(* Logix 5000 project; controller cal1615 1756-L62 rev 16.20; software revision 16.05; part 48 of 78 *)
(* tags used below, declared in another part *)
   FAULT : BOOL;   // Fault AFI
   p01_param_min_start_tension : REAL;
   p01_recipe_active : recipe;   // Active Recipe
   p01r02_plc_scan_time_in_sec : REAL;   // System PLC Scan Time in Seconds
   p01r09_pb_global_reset : BOOL;   // System Modes PB: Global Fault Reset
   p01r09_request_line_jog : BOOL;   // System Modes Request Line Jog Forward
   p01r09_stretch_mode : BOOL;
   p01r12_master_ramped_speed : REAL;   // System Line Accel Decel Control Master Ramped Speed
   p01r13_line_running : BOOL;   // System Line Start Sequence Line Running
   p01r13_line_slow_ramp : BOOL;   // System Line Start Sequence Start Line to Slow Speed
   p01r13_permissive_drives : BOOL;   // System Line Start Sequence Permissive Drives
   p01r13_state : DINT;   // System Line Start Sequence Sequencer Step
   p02_real_from_hmi : hmi_real;   // MOP HMI Iface Real from HMI
   p20r15_loa_on : BOOL;   // Letoff Letoff A VFD On
   p20r16_lob_on : BOOL;   // Letoff Letoff B On
   p22_ai_speed : REAL;
   p22_ai_ts1_lc : REAL;   // Tension Stand 1 Analog Input Loadcell
   p22_ao_selected_speed : REAL;   // Tension Stand 1 VFD Selected Speed
   p22_ao_torque : REAL;
   p22_control_word : INT;
   p22_di_brake : BOOL;   // Tension Stand 1 Digital Input Brake Temperature OK
   p22_di_jog : BOOL;   // Tension Stand 1 Digital Input SS: Jog
   p22_di_jog_fwd : BOOL;   // Tension Stand 1 Digital Input PB: Jog Forward
   p22_di_jog_rev : BOOL;   // Tension Stand 1 Digital Input PB: Jog Reverse
   p22_di_run : BOOL;   // Tension Stand 1 Digital Input SS: Run
   p22_di_therm : BOOL;   // Tension Stand 1 Digital Input Motor Temperature OK
   p22_param_ts1_jog_speed : REAL;   // System Parameter Tension Stand 1 Jog Speed
   p22_status_word : INT;
   p22_ts1_acc_rate : REAL;
   p22_ts1_decel_rate : REAL;
   p22_ts1_vfd : ABB_PROTOCOL_VFD;
   p22r01 : routine;   // Tension Stand 1 Main
   p22r02_tension_dev_max : REAL;   // Winder A VFD
   p22r02_tension_dev_min : REAL;   // Tension Stand 1 VFD
   p22r09 : routine;   // Tension Stand 1 Modes
   p22r09_mode_jog : BOOL;   // Tension Stand 1 Modes Jog Mode
   p22r09_mode_run : BOOL;   // Tension Stand 1 Modes Run Mode
   p22r09_mode_thread : BOOL;   // Tension Stand 1 Modes Thread Mode
   p22r09_pb_jog_fwd : BOOL;   // Tension Stand 1 Modes PB: Jog Forward
   p22r09_pb_jog_rev : BOOL;   // Tension Stand 1 Modes PB: Jog Reverse
   p22r09_timer_fault : TIMER[4];   // Tension Stand 1 Modes Fault Delay
   p22r09_timer_warning : TIMER[4];   // Tension Stand 1 Modes Warning Delay
   p22r10 : routine;   // Tension Stand 1 Speed Tension
   p22r10_calc_speed_offset : REAL;
   p22r10_param_psn_gain : REAL;   // Tension Stand 1 Parameter Position Gain
   p22r10_pid_out : REAL;
   p22r10_pid_psn : PID;   // Tension Stand 1 Speed Tension PID Dancer Position
   p22r10_pid_psn_cv : REAL;   // Tension Stand 1 Speed Tension PID Dancer Position Control Variable
   p22r10_pid_psn_pv : REAL;   // Tension Stand 1 Speed Tension PID Dancer Position Process Variable
   p22r10_selected_torque : REAL;
   p22r10_speed_offset : REAL;   // Tension Stand 1 Speed tension Speed Offset from Base
   p22r10_stretch : REAL;
   p22r10_timer_fault : TIMER[4];   // Tension Stand 1 Speed Tension Fault Delay
   p22r10_timer_warning : TIMER[4];   // Tension Stand 1 Speed Tension Warning Delay
   p22r11 : routine;   // Tension Stand 1 VFD
   p22r11_acc_decel_ramp : SYS_ACC_DEC_RAMP;   // Tension Stand 1 VFD Accel/Decel Ramp
   p22r11_permissive_jog : BOOL;   // Tension Stand 1 VFD Permissive Run
   p22r11_request_jog_fwd : BOOL;   // Tension Stand 1 VFD Request Jog FWD
   p22r11_request_jog_rev : BOOL;   // Tension Stand 1 VFD Request Jog REV
   p22r11_request_line_jog : BOOL;   // Tension Stand 1 VFD Request Line Jog
   p22r11_request_line_run : BOOL;   // Tension Stant 1 VFD Request Line Run
   p22r11_request_start : BOOL;   // Tension Stand 1 VFD
   p22r11_request_tension : BOOL;
   p22r11_request_thread_fwd : BOOL;   // Tension Stand 1 VFD Request Thread FWD
   p22r11_request_thread_rev : BOOL;   // Tension Stand 1 VFD Request Thread REV
   p22r11_selected_speed : REAL;   // Tension Stand 1 VFD Selected Speed
   p22r11_timer_fault : TIMER[10];   // Tension Stand 1 VFD Fault Timer
   p22r11_timer_warning : TIMER[5];   // Tension Stand 1 VFD Warning Timer
   p22r11_zero_speed : BOOL;   // Tension Stand 1 VFD Zero Speed
   p23r15_pid_tension_control : BOOL;   // Impreg Metering Roll VFD PID Wet Web Active
   p25r09_mode_thread : BOOL;   // Tension Stand 2 Modes Thread Mode
   p25r09_pb_jog_fwd : BOOL;   // Tension Stand 2 Modes PB: Jog Forward
   p25r09_pb_jog_rev : BOOL;   // Tension Stand 2 Modes PB: Jog Reverse
(* P22_Tension_Stand_1, continued *)

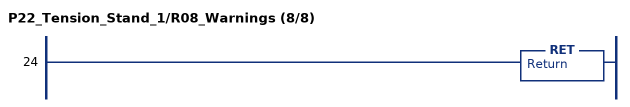
   [picture p936: P22_Tension_Stand_1/R08_Warnings rungs 24-24]
   24: RET();
END_ROUTINE

ROUTINE R09_Modes   (* ladder *)
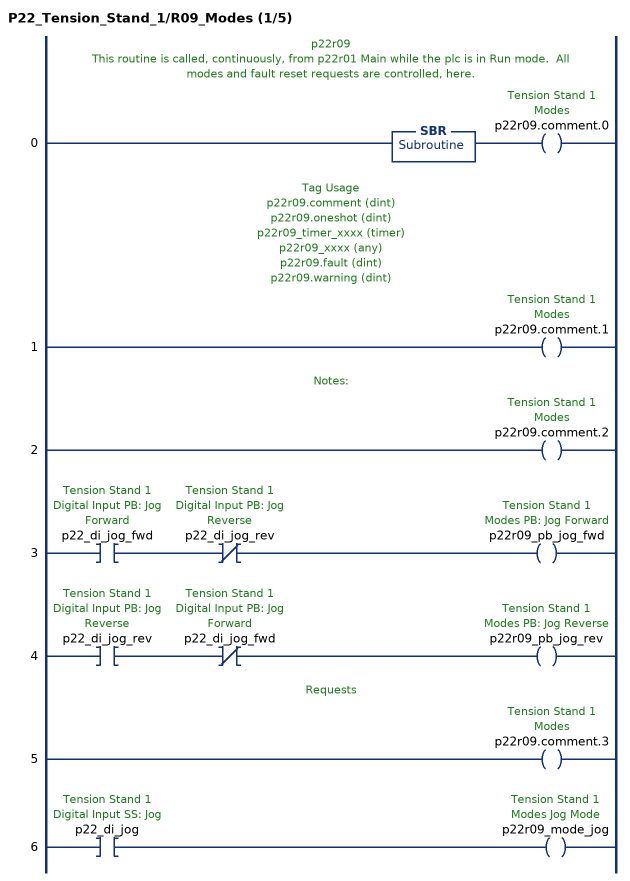
   // p22r09
   // This routine is called, continuously, from p22r01 Main while the plc is in Run mode.  All modes and fault reset requests are controlled, here.
   0: SBR()OTE(p22r09.comment.0);
   // Tag Usage
   // p22r09.comment (dint)
   // p22r09.oneshot (dint)
   // p22r09_timer_xxxx (timer)
   // p22r09_xxxx (any)
   // p22r09.fault (dint)
   // p22r09.warning (dint)
   1: OTE(p22r09.comment.1);
   // Notes:
   2: OTE(p22r09.comment.2);
   3: XIC(p22_di_jog_fwd)XIO(p22_di_jog_rev)OTE(p22r09_pb_jog_fwd);
   4: XIC(p22_di_jog_rev)XIO(p22_di_jog_fwd)OTE(p22r09_pb_jog_rev);
   // Requests
   5: OTE(p22r09.comment.3);
   6: XIC(p22_di_jog)OTE(p22r09_mode_jog);
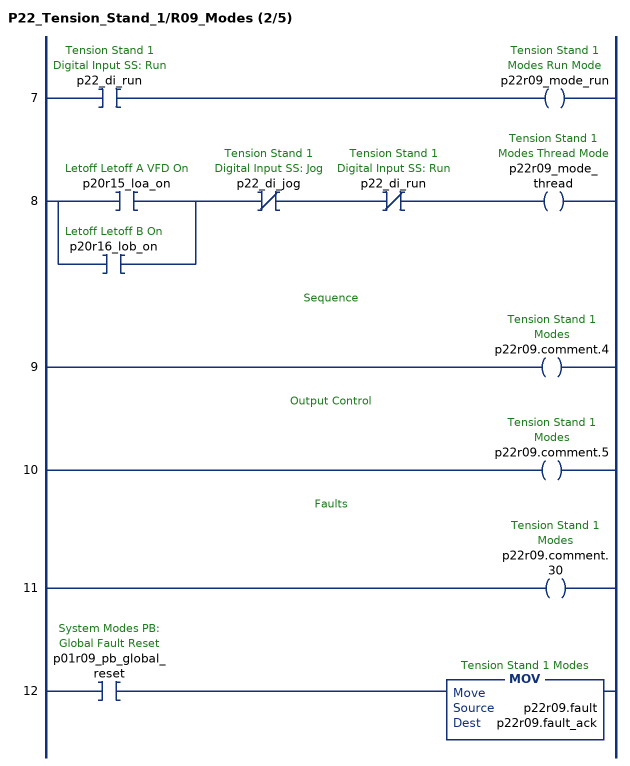
   7: XIC(p22_di_run)OTE(p22r09_mode_run);
   8: [XIC(p20r15_loa_on) ,XIC(p20r16_lob_on) ]XIO(p22_di_jog)XIO(p22_di_run)OTE(p22r09_mode_thread);
   // Sequence
   9: OTE(p22r09.comment.4);
   // Output Control
   10: OTE(p22r09.comment.5);
   // Faults
   11: OTE(p22r09.comment.30);
   12: XIC(p01r09_pb_global_reset)MOV(p22r09.fault,p22r09.fault_ack);
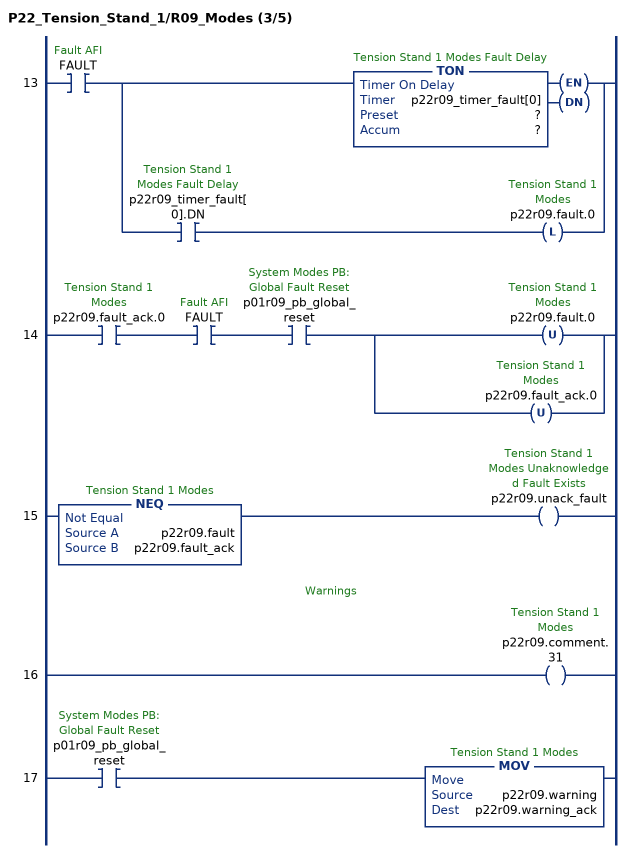
   13: XIC(FAULT)[TON(p22r09_timer_fault[0],?,?) ,XIC(p22r09_timer_fault[0].DN) OTL(p22r09.fault.0) ];
   14: XIC(p22r09.fault_ack.0)XIC(FAULT)XIC(p01r09_pb_global_reset)[OTU(p22r09.fault.0) ,OTU(p22r09.fault_ack.0) ];
   15: NEQ(p22r09.fault,p22r09.fault_ack)OTE(p22r09.unack_fault);
   // Warnings
   16: OTE(p22r09.comment.31);
   17: XIC(p01r09_pb_global_reset)MOV(p22r09.warning,p22r09.warning_ack);
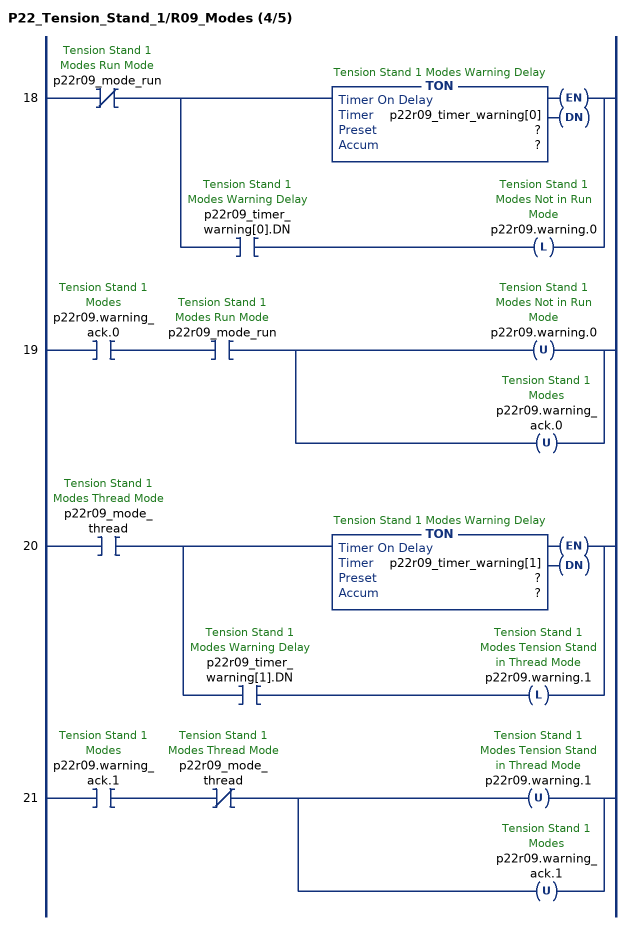
   18: XIO(p22r09_mode_run)[TON(p22r09_timer_warning[0],?,?) ,XIC(p22r09_timer_warning[0].DN) OTL(p22r09.warning.0) ];
   19: XIC(p22r09.warning_ack.0)XIC(p22r09_mode_run)[OTU(p22r09.warning.0) ,OTU(p22r09.warning_ack.0) ];
   20: XIC(p22r09_mode_thread)[TON(p22r09_timer_warning[1],?,?) ,XIC(p22r09_timer_warning[1].DN) OTL(p22r09.warning.1) ];
   21: XIC(p22r09.warning_ack.1)XIO(p22r09_mode_thread)[OTU(p22r09.warning.1) ,OTU(p22r09.warning_ack.1) ];
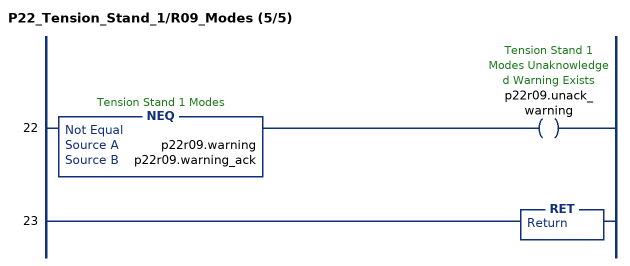
   22: NEQ(p22r09.warning,p22r09.warning_ack)OTE(p22r09.unack_warning);
   23: RET();
END_ROUTINE

ROUTINE R10_Speed_Control   (* ladder *)
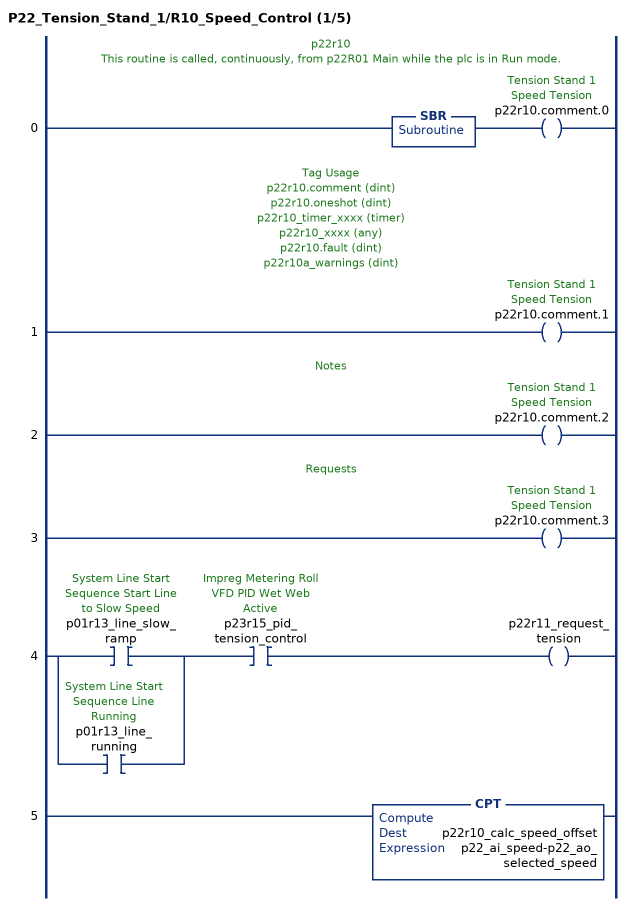
   // p22r10
   // This routine is called, continuously, from p22R01 Main while the plc is in Run mode.
   0: SBR()OTE(p22r10.comment.0);
   // Tag Usage
   // p22r10.comment (dint)
   // p22r10.oneshot (dint)
   // p22r10_timer_xxxx (timer)
   // p22r10_xxxx (any)
   // p22r10.fault (dint)
   // p22r10a_warnings (dint)
   1: OTE(p22r10.comment.1);
   // Notes
   2: OTE(p22r10.comment.2);
   // Requests
   3: OTE(p22r10.comment.3);
   4: [XIC(p01r13_line_slow_ramp) ,XIC(p01r13_line_running) ]XIC(p23r15_pid_tension_control)OTE(p22r11_request_tension);
   5: CPT(p22r10_calc_speed_offset,p22_ai_speed-p22_ao_selected_speed);
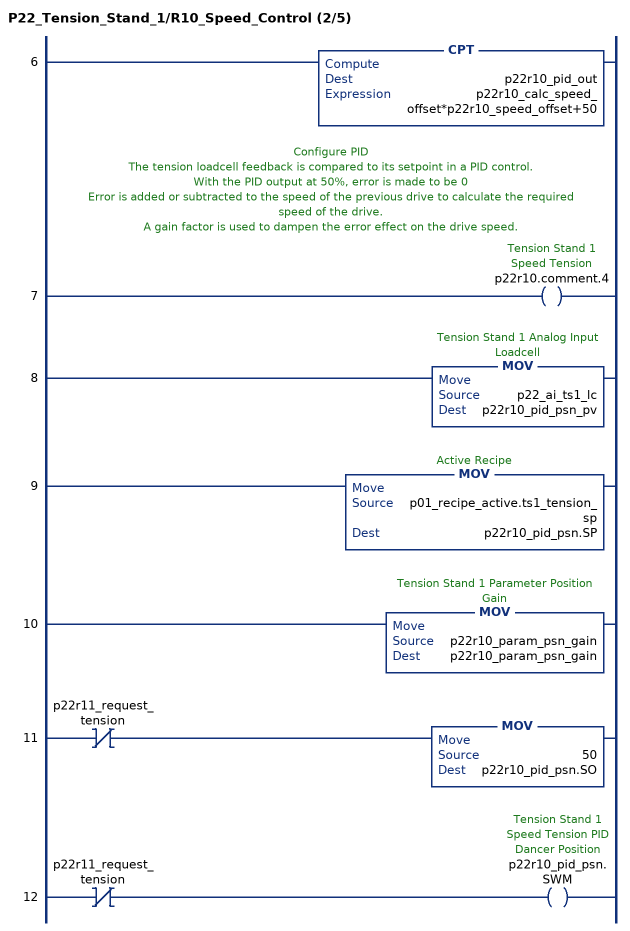
   6: CPT(p22r10_pid_out,p22r10_calc_speed_offset*p22r10_speed_offset+50);
   // Configure PID
   // The tension loadcell feedback is compared to its setpoint in a PID control.
   // With the PID output at 50%, error is made to be 0
   // Error is added or subtracted to the speed of the previous drive to calculate the required speed of the drive.
   // A gain factor is used to dampen the error effect on the drive speed.
   7: OTE(p22r10.comment.4);
   8: MOV(p22_ai_ts1_lc,p22r10_pid_psn_pv);
   9: MOV(p01_recipe_active.ts1_tension_sp,p22r10_pid_psn.SP);
   10: MOV(p22r10_param_psn_gain,p22r10_param_psn_gain);
   11: XIO(p22r11_request_tension)MOV(50,p22r10_pid_psn.SO);
   12: XIO(p22r11_request_tension)OTE(p22r10_pid_psn.SWM);
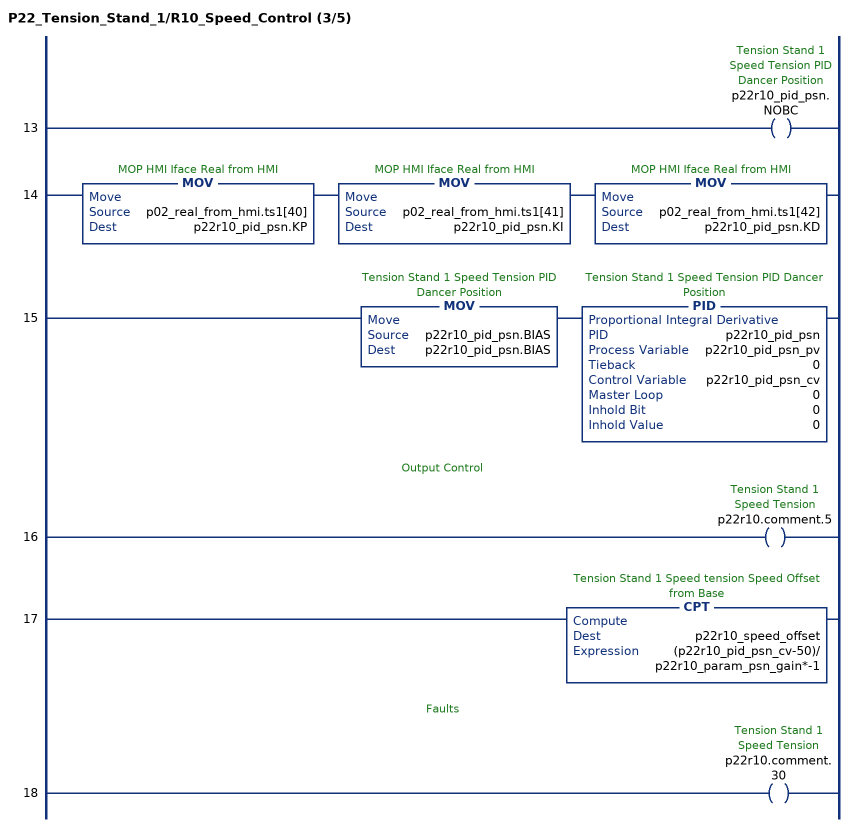
   13: OTE(p22r10_pid_psn.NOBC);
   14: MOV(p02_real_from_hmi.ts1[40],p22r10_pid_psn.KP)MOV(p02_real_from_hmi.ts1[41],p22r10_pid_psn.KI)MOV(p02_real_from_hmi.ts1[42],p22r10_pid_psn.KD);
   15: MOV(p22r10_pid_psn.BIAS,p22r10_pid_psn.BIAS)PID(p22r10_pid_psn,p22r10_pid_psn_pv,0,p22r10_pid_psn_cv,0,0,0);
   // Output Control
   16: OTE(p22r10.comment.5);
   17: CPT(p22r10_speed_offset,(p22r10_pid_psn_cv-50)/p22r10_param_psn_gain*-1);
   // Faults
   18: OTE(p22r10.comment.30);
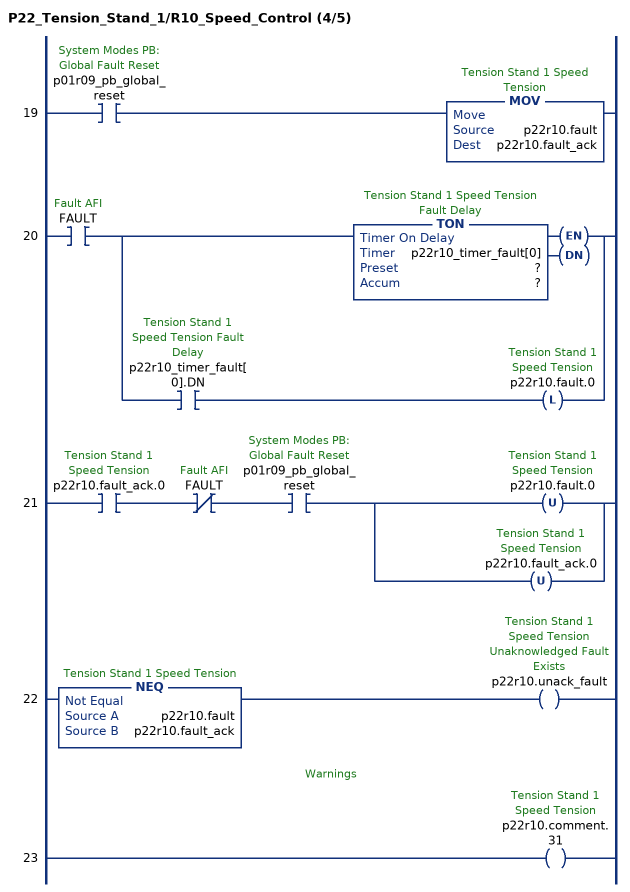
   19: XIC(p01r09_pb_global_reset)MOV(p22r10.fault,p22r10.fault_ack);
   20: XIC(FAULT)[TON(p22r10_timer_fault[0],?,?) ,XIC(p22r10_timer_fault[0].DN) OTL(p22r10.fault.0) ];
   21: XIC(p22r10.fault_ack.0)XIO(FAULT)XIC(p01r09_pb_global_reset)[OTU(p22r10.fault.0) ,OTU(p22r10.fault_ack.0) ];
   22: NEQ(p22r10.fault,p22r10.fault_ack)OTE(p22r10.unack_fault);
   // Warnings
   23: OTE(p22r10.comment.31);
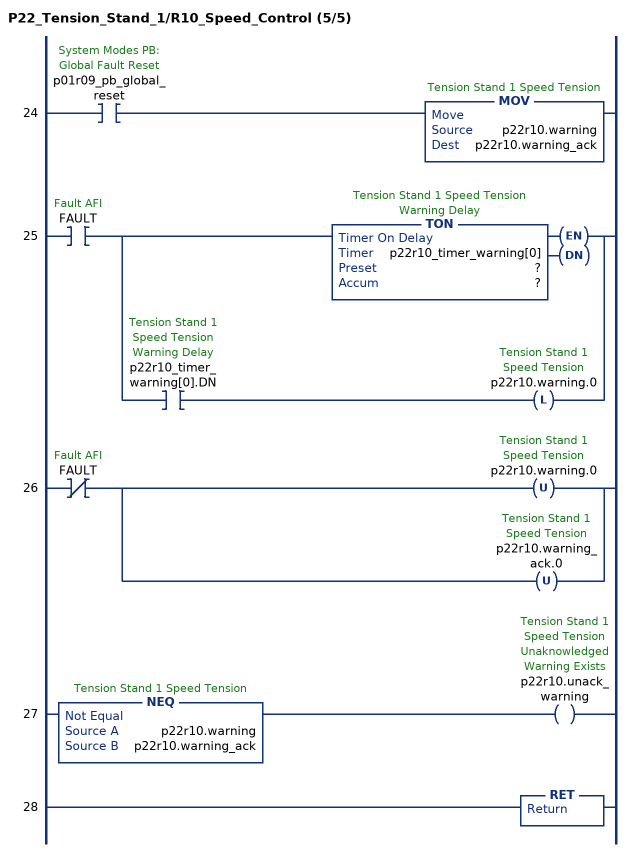
   24: XIC(p01r09_pb_global_reset)MOV(p22r10.warning,p22r10.warning_ack);
   25: XIC(FAULT)[TON(p22r10_timer_warning[0],?,?) ,XIC(p22r10_timer_warning[0].DN) OTL(p22r10.warning.0) ];
   26: XIO(FAULT)[OTU(p22r10.warning.0) ,OTU(p22r10.warning_ack.0) ];
   27: NEQ(p22r10.warning,p22r10.warning_ack)OTE(p22r10.unack_warning);
   28: RET();
END_ROUTINE

ROUTINE R11_VFD   (* ladder *)
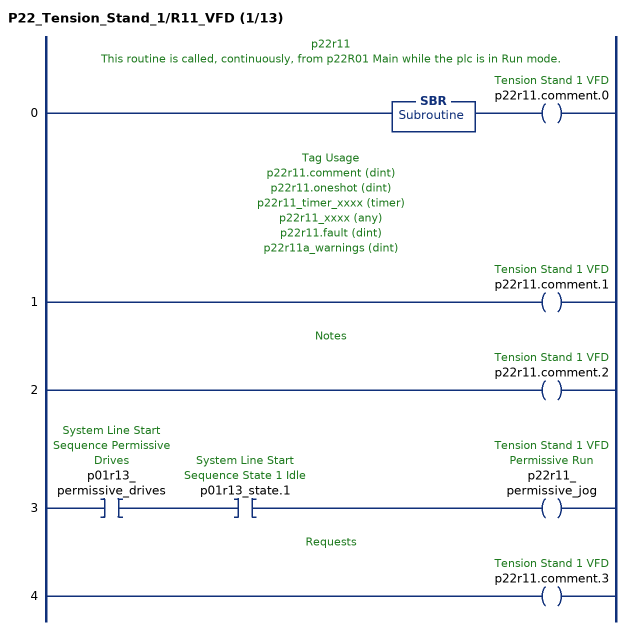
   // p22r11
   // This routine is called, continuously, from p22R01 Main while the plc is in Run mode.
   0: SBR()OTE(p22r11.comment.0);
   // Tag Usage
   // p22r11.comment (dint)
   // p22r11.oneshot (dint)
   // p22r11_timer_xxxx (timer)
   // p22r11_xxxx (any)
   // p22r11.fault (dint)
   // p22r11a_warnings (dint)
   1: OTE(p22r11.comment.1);
   // Notes
   2: OTE(p22r11.comment.2);
   3: XIC(p01r13_permissive_drives)XIC(p01r13_state.1)OTE(p22r11_permissive_jog);
   // Requests
   4: OTE(p22r11.comment.3);
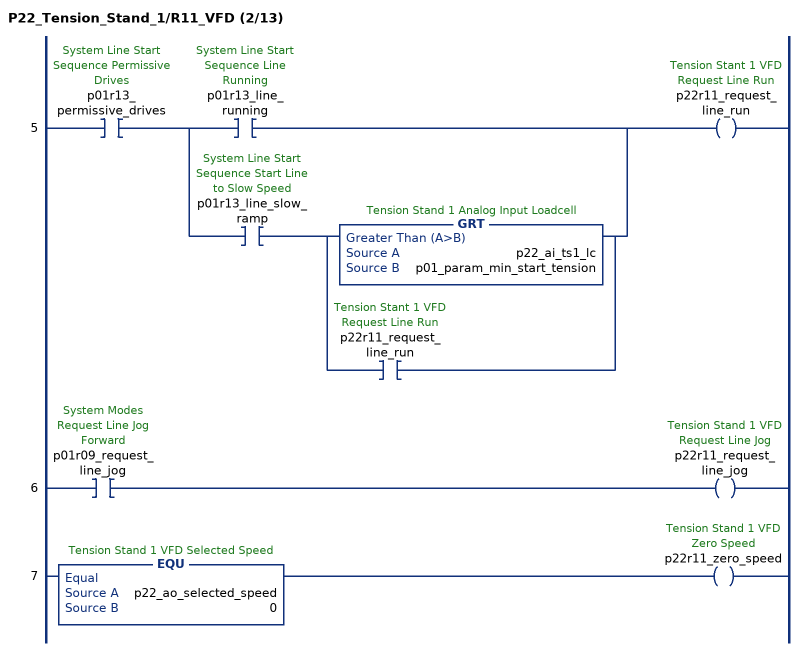
   5: XIC(p01r13_permissive_drives)[XIC(p01r13_line_running) ,XIC(p01r13_line_slow_ramp) [GRT(p22_ai_ts1_lc,p01_param_min_start_tension) ,XIC(p22r11_request_line_run) ] ]OTE(p22r11_request_line_run);
   6: XIC(p01r09_request_line_jog)OTE(p22r11_request_line_jog);
   7: EQU(p22_ao_selected_speed,0)OTE(p22r11_zero_speed);
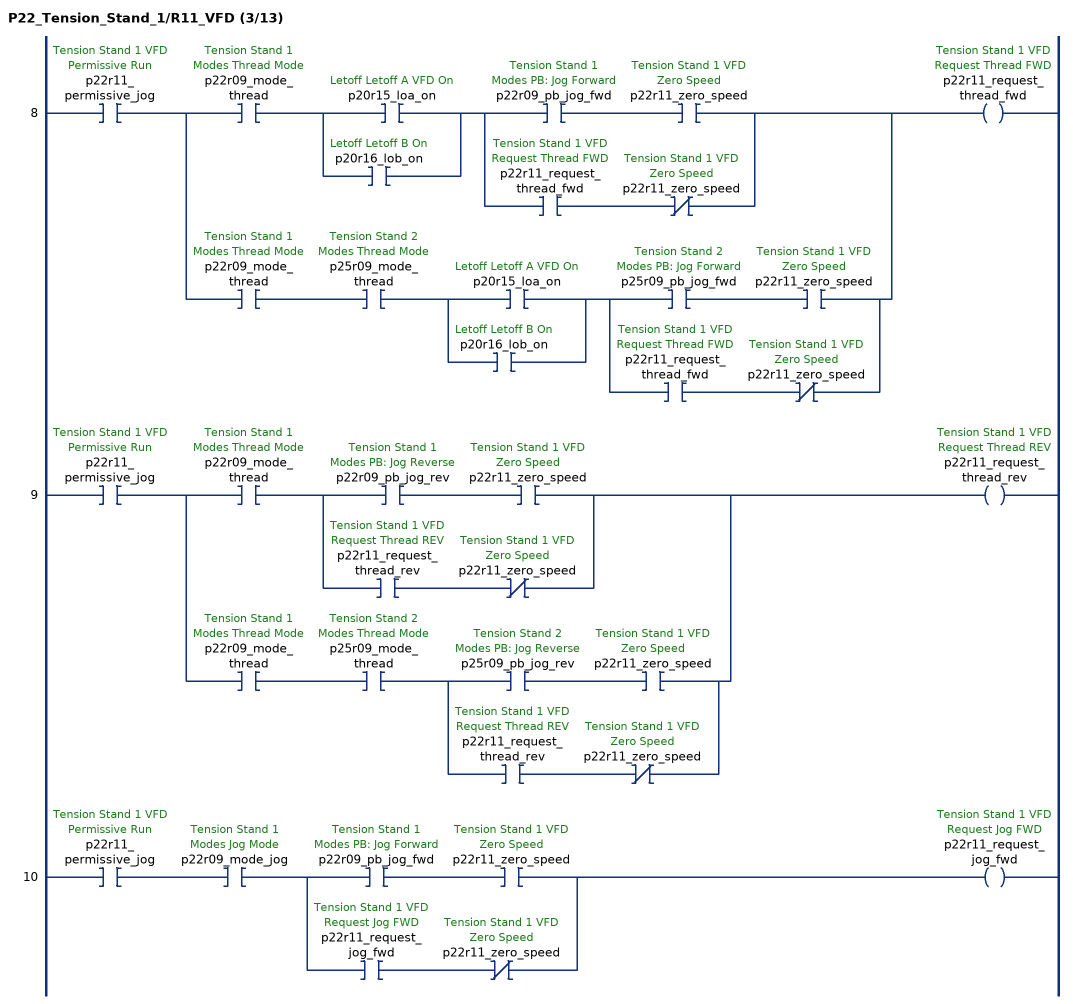
   8: XIC(p22r11_permissive_jog)[XIC(p22r09_mode_thread) [XIC(p20r15_loa_on) ,XIC(p20r16_lob_on) ] [XIC(p22r09_pb_jog_fwd) XIC(p22r11_zero_speed) ,XIC(p22r11_request_thread_fwd) XIO(p22r11_zero_speed) ] ,XIC(p22r09_mode_thread) XIC(p25r09_mode_thread) [XIC(p20r15_loa_on) ,XIC(p20r16_lob_on) ] [XIC(p25r09_pb_jog_fwd) XIC(p22r11_zero_speed) ,XIC(p22r11_request_thread_fwd) XIO(p22r11_zero_speed) ] ]OTE(p22r11_request_thread_fwd);
   9: XIC(p22r11_permissive_jog)[XIC(p22r09_mode_thread) [XIC(p22r09_pb_jog_rev) XIC(p22r11_zero_speed) ,XIC(p22r11_request_thread_rev) XIO(p22r11_zero_speed) ] ,XIC(p22r09_mode_thread) XIC(p25r09_mode_thread) [XIC(p25r09_pb_jog_rev) XIC(p22r11_zero_speed) ,XIC(p22r11_request_thread_rev) XIO(p22r11_zero_speed) ] ]OTE(p22r11_request_thread_rev);
   10: XIC(p22r11_permissive_jog)XIC(p22r09_mode_jog)[XIC(p22r09_pb_jog_fwd) XIC(p22r11_zero_speed) ,XIC(p22r11_request_jog_fwd) XIO(p22r11_zero_speed) ]OTE(p22r11_request_jog_fwd);
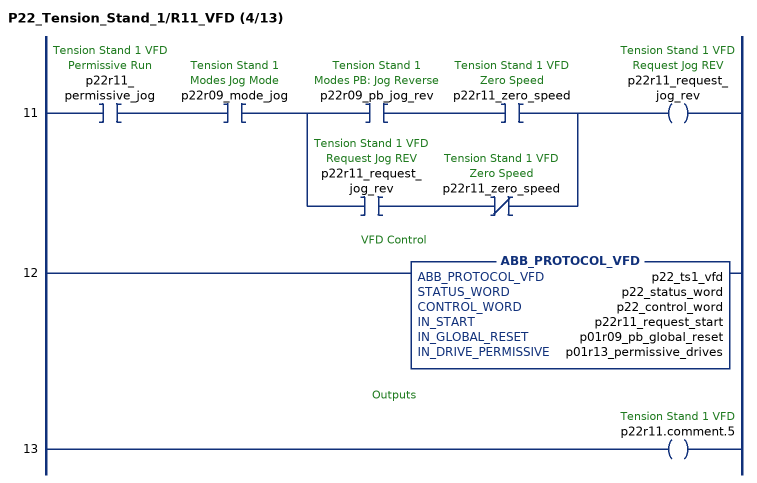
   11: XIC(p22r11_permissive_jog)XIC(p22r09_mode_jog)[XIC(p22r09_pb_jog_rev) XIC(p22r11_zero_speed) ,XIC(p22r11_request_jog_rev) XIO(p22r11_zero_speed) ]OTE(p22r11_request_jog_rev);
   // VFD Control
   12: ABB_PROTOCOL_VFD(p22_ts1_vfd,p22_status_word,p22_control_word,p22r11_request_start,p01r09_pb_global_reset,p01r13_permissive_drives);
   // Outputs
   13: OTE(p22r11.comment.5);
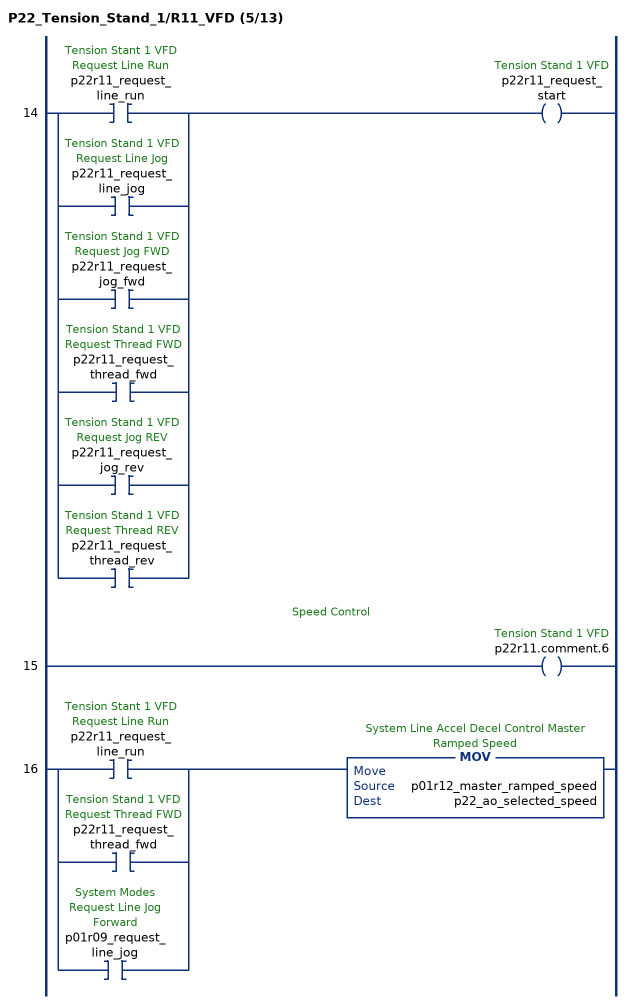
   14: [XIC(p22r11_request_line_run) ,XIC(p22r11_request_line_jog) ,XIC(p22r11_request_jog_fwd) ,XIC(p22r11_request_thread_fwd) ,XIC(p22r11_request_jog_rev) ,XIC(p22r11_request_thread_rev) ]OTE(p22r11_request_start);
   // Speed Control
   15: OTE(p22r11.comment.6);
   16: [XIC(p22r11_request_line_run) ,XIC(p22r11_request_thread_fwd) ,XIC(p01r09_request_line_jog) ]MOV(p01r12_master_ramped_speed,p22_ao_selected_speed);
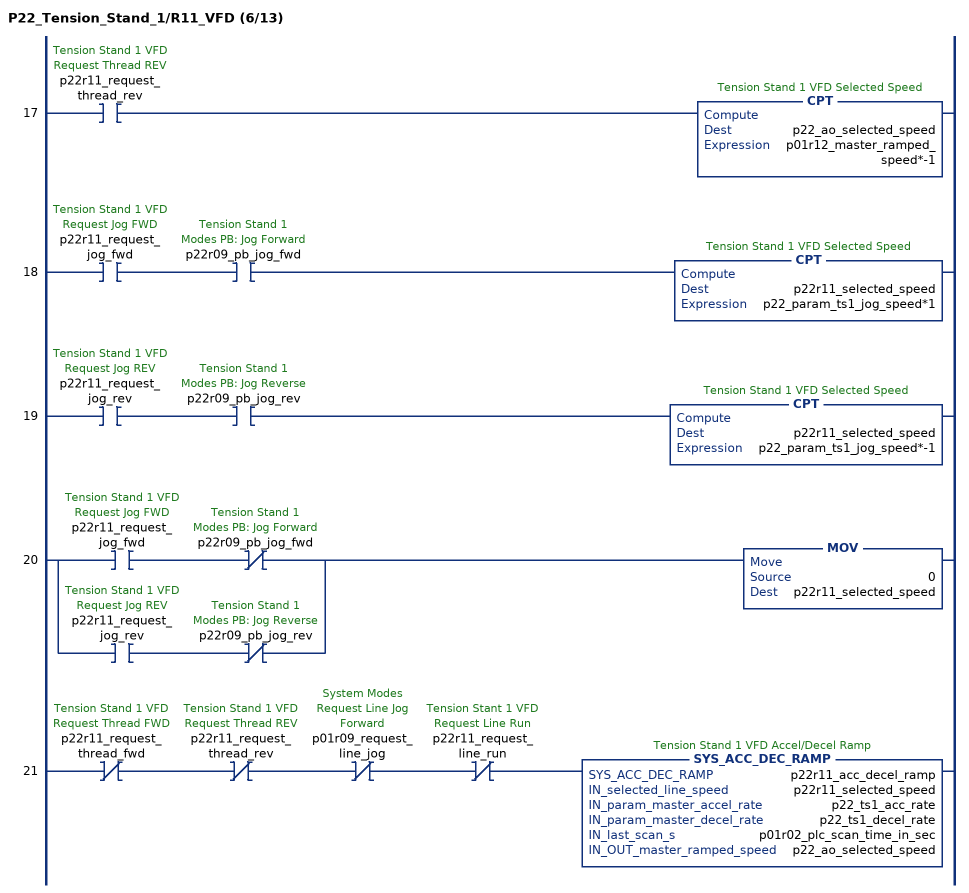
   17: XIC(p22r11_request_thread_rev)CPT(p22_ao_selected_speed,p01r12_master_ramped_speed*-1);
   18: XIC(p22r11_request_jog_fwd)XIC(p22r09_pb_jog_fwd)CPT(p22r11_selected_speed,p22_param_ts1_jog_speed*1);
   19: XIC(p22r11_request_jog_rev)XIC(p22r09_pb_jog_rev)CPT(p22r11_selected_speed,p22_param_ts1_jog_speed*-1);
   20: [XIC(p22r11_request_jog_fwd) XIO(p22r09_pb_jog_fwd) ,XIC(p22r11_request_jog_rev) XIO(p22r09_pb_jog_rev) ]MOV(0,p22r11_selected_speed);
   21: XIO(p22r11_request_thread_fwd)XIO(p22r11_request_thread_rev)XIO(p01r09_request_line_jog)XIO(p22r11_request_line_run)SYS_ACC_DEC_RAMP(p22r11_acc_decel_ramp,p22r11_selected_speed,p22_ts1_acc_rate,p22_ts1_decel_rate,p01r02_plc_scan_time_in_sec,p22_ao_selected_speed);
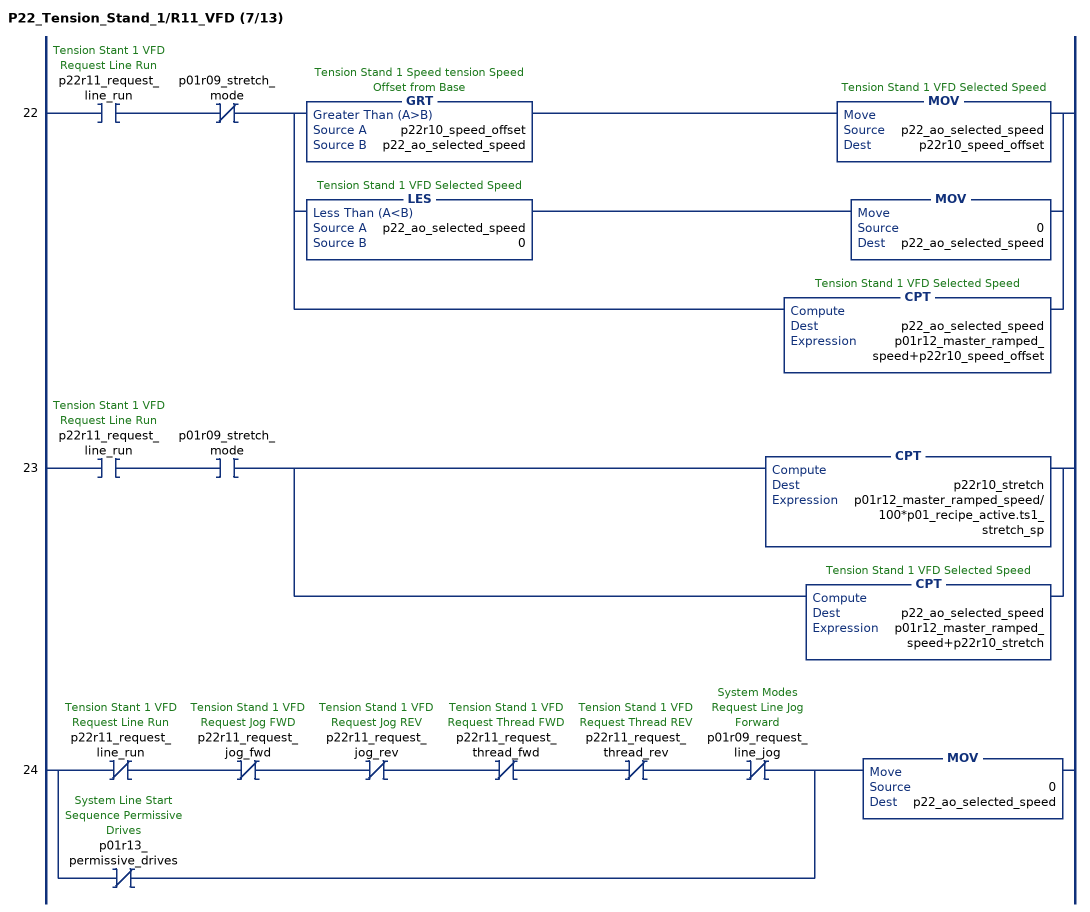
   22: XIC(p22r11_request_line_run)XIO(p01r09_stretch_mode)[GRT(p22r10_speed_offset,p22_ao_selected_speed) MOV(p22_ao_selected_speed,p22r10_speed_offset) ,LES(p22_ao_selected_speed,0) MOV(0,p22_ao_selected_speed) ,CPT(p22_ao_selected_speed,p01r12_master_ramped_speed+p22r10_speed_offset) ];
   23: XIC(p22r11_request_line_run)XIC(p01r09_stretch_mode)[CPT(p22r10_stretch,p01r12_master_ramped_speed/100*p01_recipe_active.ts1_stretch_sp) ,CPT(p22_ao_selected_speed,p01r12_master_ramped_speed+p22r10_stretch) ];
   24: [XIO(p22r11_request_line_run) XIO(p22r11_request_jog_fwd) XIO(p22r11_request_jog_rev) XIO(p22r11_request_thread_fwd) XIO(p22r11_request_thread_rev) XIO(p01r09_request_line_jog) ,XIO(p01r13_permissive_drives) ]MOV(0,p22_ao_selected_speed);
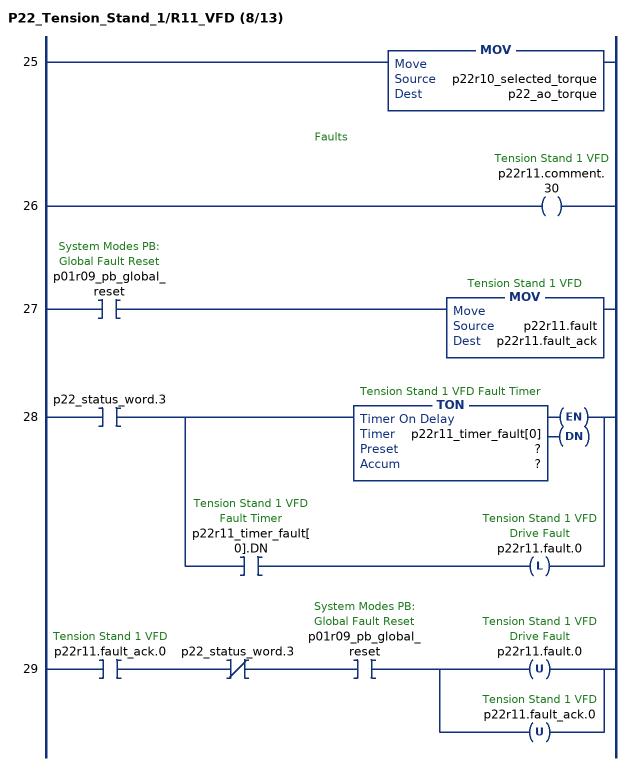
   25: MOV(p22r10_selected_torque,p22_ao_torque);
   // Faults
   26: OTE(p22r11.comment.30);
   27: XIC(p01r09_pb_global_reset)MOV(p22r11.fault,p22r11.fault_ack);
   28: XIC(p22_status_word.3)[TON(p22r11_timer_fault[0],?,?) ,XIC(p22r11_timer_fault[0].DN) OTL(p22r11.fault.0) ];
   29: XIC(p22r11.fault_ack.0)XIO(p22_status_word.3)XIC(p01r09_pb_global_reset)[OTU(p22r11.fault.0) ,OTU(p22r11.fault_ack.0) ];
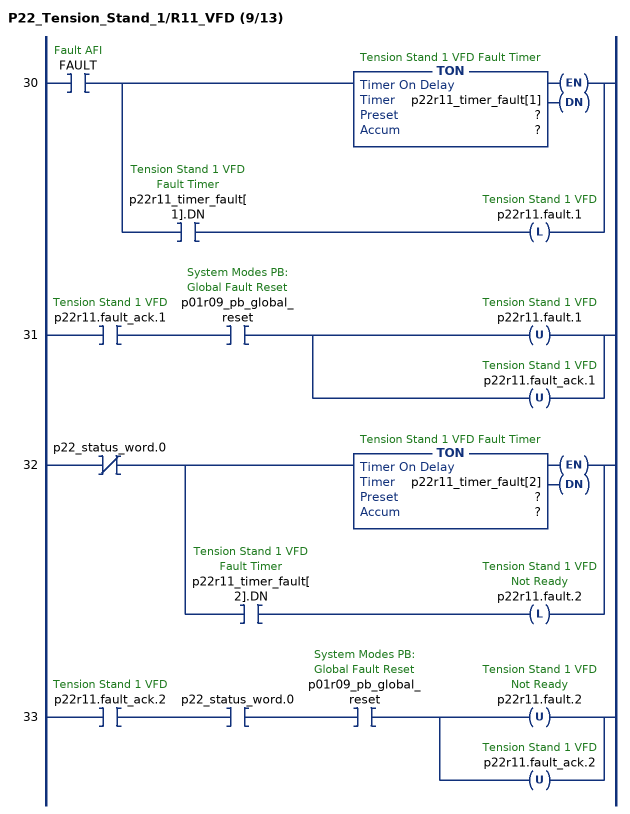
   30: XIC(FAULT)[TON(p22r11_timer_fault[1],?,?) ,XIC(p22r11_timer_fault[1].DN) OTL(p22r11.fault.1) ];
   31: XIC(p22r11.fault_ack.1)XIC(p01r09_pb_global_reset)[OTU(p22r11.fault.1) ,OTU(p22r11.fault_ack.1) ];
   32: XIO(p22_status_word.0)[TON(p22r11_timer_fault[2],?,?) ,XIC(p22r11_timer_fault[2].DN) OTL(p22r11.fault.2) ];
   33: XIC(p22r11.fault_ack.2)XIC(p22_status_word.0)XIC(p01r09_pb_global_reset)[OTU(p22r11.fault.2) ,OTU(p22r11.fault_ack.2) ];
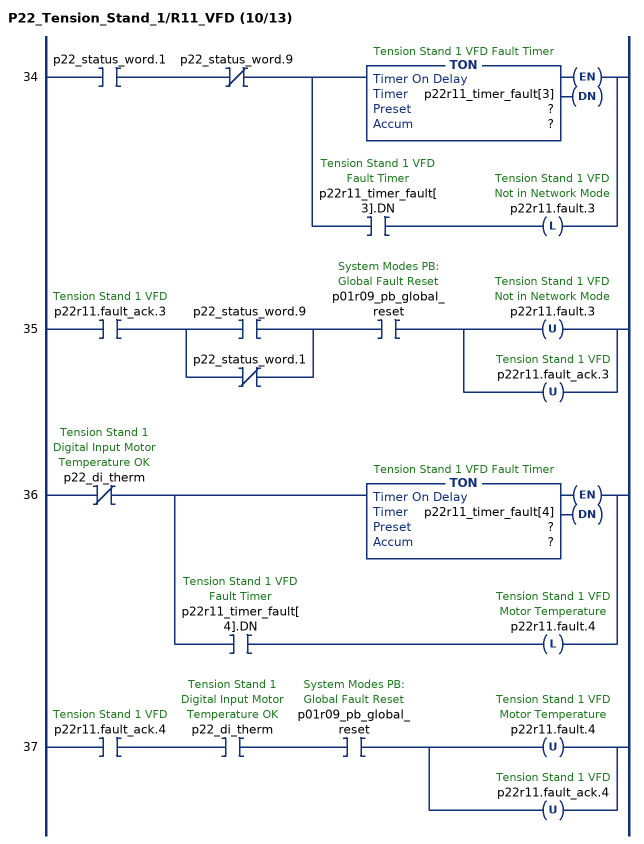
   34: XIC(p22_status_word.1)XIO(p22_status_word.9)[TON(p22r11_timer_fault[3],?,?) ,XIC(p22r11_timer_fault[3].DN) OTL(p22r11.fault.3) ];
   35: XIC(p22r11.fault_ack.3)[XIC(p22_status_word.9) ,XIO(p22_status_word.1) ]XIC(p01r09_pb_global_reset)[OTU(p22r11.fault.3) ,OTU(p22r11.fault_ack.3) ];
   36: XIO(p22_di_therm)[TON(p22r11_timer_fault[4],?,?) ,XIC(p22r11_timer_fault[4].DN) OTL(p22r11.fault.4) ];
   37: XIC(p22r11.fault_ack.4)XIC(p22_di_therm)XIC(p01r09_pb_global_reset)[OTU(p22r11.fault.4) ,OTU(p22r11.fault_ack.4) ];
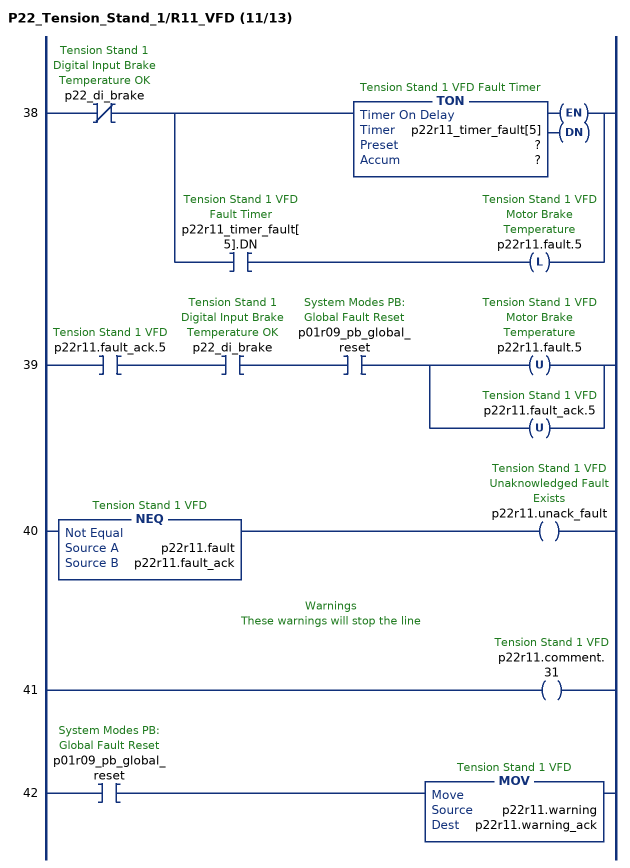
   38: XIO(p22_di_brake)[TON(p22r11_timer_fault[5],?,?) ,XIC(p22r11_timer_fault[5].DN) OTL(p22r11.fault.5) ];
   39: XIC(p22r11.fault_ack.5)XIC(p22_di_brake)XIC(p01r09_pb_global_reset)[OTU(p22r11.fault.5) ,OTU(p22r11.fault_ack.5) ];
   40: NEQ(p22r11.fault,p22r11.fault_ack)OTE(p22r11.unack_fault);
   // Warnings
   // These warnings will stop the line
   41: OTE(p22r11.comment.31);
   42: XIC(p01r09_pb_global_reset)MOV(p22r11.warning,p22r11.warning_ack);
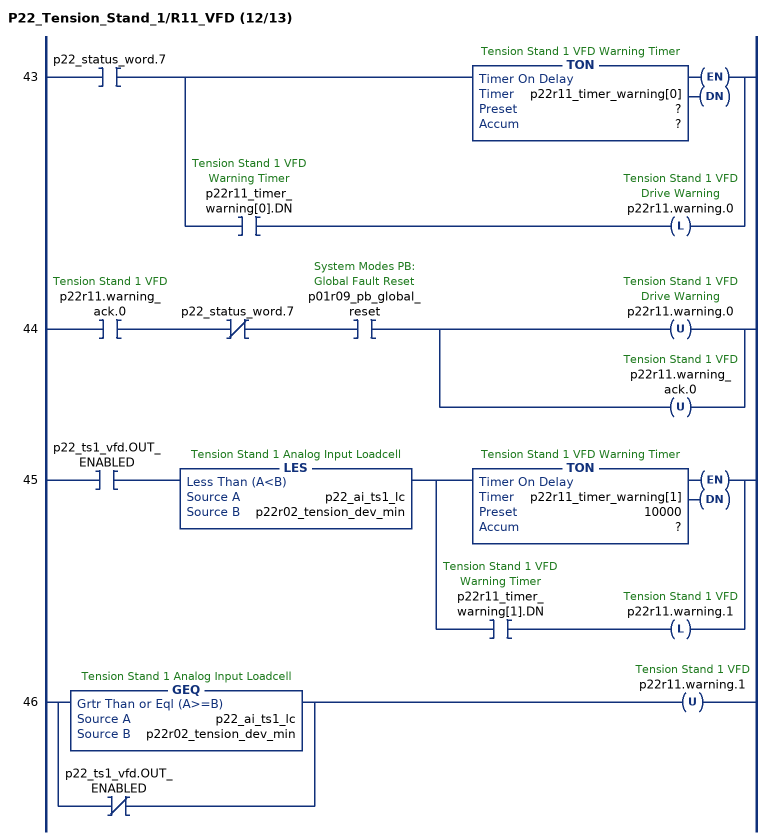
   43: XIC(p22_status_word.7)[TON(p22r11_timer_warning[0],?,?) ,XIC(p22r11_timer_warning[0].DN) OTL(p22r11.warning.0) ];
   44: XIC(p22r11.warning_ack.0)XIO(p22_status_word.7)XIC(p01r09_pb_global_reset)[OTU(p22r11.warning.0) ,OTU(p22r11.warning_ack.0) ];
   45: XIC(p22_ts1_vfd.OUT_ENABLED)LES(p22_ai_ts1_lc,p22r02_tension_dev_min)[TON(p22r11_timer_warning[1],?,?) ,XIC(p22r11_timer_warning[1].DN) OTL(p22r11.warning.1) ];
   46: [GEQ(p22_ai_ts1_lc,p22r02_tension_dev_min) ,XIO(p22_ts1_vfd.OUT_ENABLED) ]OTU(p22r11.warning.1);
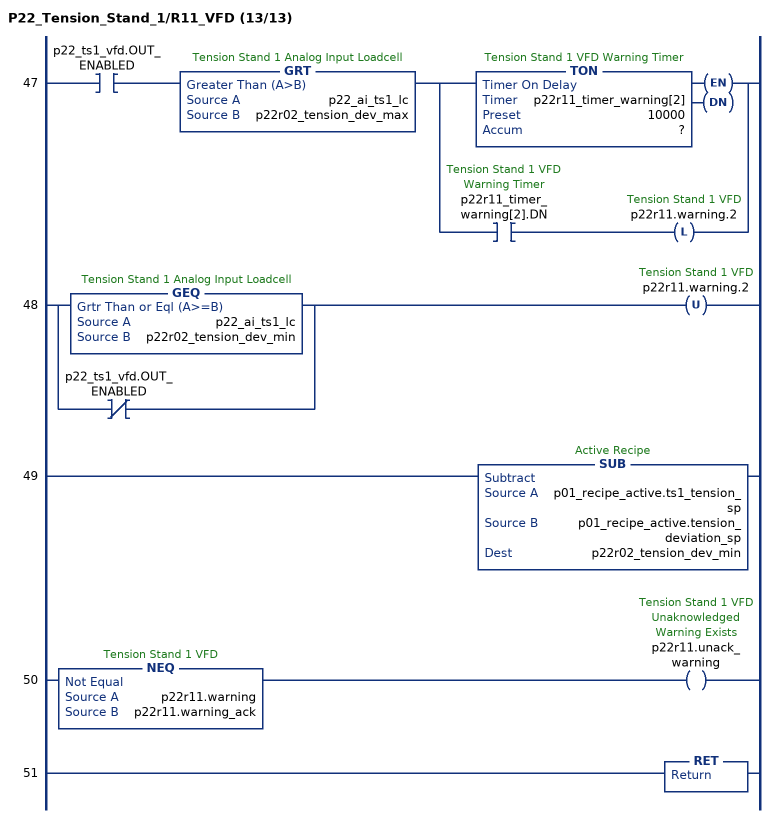
   47: XIC(p22_ts1_vfd.OUT_ENABLED)GRT(p22_ai_ts1_lc,p22r02_tension_dev_max)[TON(p22r11_timer_warning[2],?,?) ,XIC(p22r11_timer_warning[2].DN) OTL(p22r11.warning.2) ];
   48: [GEQ(p22_ai_ts1_lc,p22r02_tension_dev_min) ,XIO(p22_ts1_vfd.OUT_ENABLED) ]OTU(p22r11.warning.2);
   49: SUB(p01_recipe_active.ts1_tension_sp,p01_recipe_active.tension_deviation_sp,p22r02_tension_dev_min);
   50: NEQ(p22r11.warning,p22r11.warning_ack)OTE(p22r11.unack_warning);
   51: RET();
END_ROUTINE
END_PROGRAM
